FUNCTION_BLOCK Port (* Service Interface Function Block Type *)
  (* Standard: 61499-2; Description: Copyright (c) 2021, 2022 Jonathan Lainer This program and the accompanying materials are made available under the terms of the Eclipse Public License 2.0 which is available at https://www.eclipse.org/legal/epl-2.0/ SPDX-License-Identifier: EPL-2.0 *)
  (* Version 3.0, 2025-04-14, Patrick Aigner, changed package *)
  (* Version 1.0, 2021-02-22, Jonathan Lainer, Initial Contribution *)
  PACKAGE eclipse4diac::io::eliteboard;
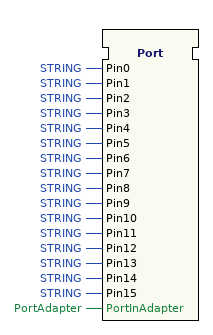
  VAR_INPUT
    Pin0 : STRING; (* Name of the Pin *)
    Pin1 : STRING; (* Name of the Pin *)
    Pin2 : STRING; (* Name of the Pin *)
    Pin3 : STRING; (* Name of the Pin *)
    Pin4 : STRING; (* Name of the Pin *)
    Pin5 : STRING; (* Name of the Pin *)
    Pin6 : STRING; (* Name of the Pin *)
    Pin7 : STRING; (* Name of the Pin *)
    Pin8 : STRING; (* Name of the Pin *)
    Pin9 : STRING; (* Name of the Pin *)
    Pin10 : STRING; (* Name of the Pin *)
    Pin11 : STRING; (* Name of the Pin *)
    Pin12 : STRING; (* Name of the Pin *)
    Pin13 : STRING; (* Name of the Pin *)
    Pin14 : STRING; (* Name of the Pin *)
    Pin15 : STRING; (* Name of the Pin *)
  END_VAR
  SOCKETS
    PortInAdapter : eclipse4diac::io::eliteboard::PortAdapter;
  END_SOCKETS
END_FUNCTION_BLOCK
